Fanuc TP program (LS listing): set_pass_sr.ls

/PROG  SET_PASS_SR
/ATTR
OWNER		= MNEDITOR;
COMMENT		= "";
PROG_SIZE	= 148;
CREATE		= DATE 25-08-01  TIME 09:50:32;
MODIFIED	= DATE 25-08-01  TIME 09:50:32;
FILE_NAME	= ;
VERSION		= 0;
LINE_COUNT	= 1;
MEMORY_SIZE	= 516;
PROTECT		= READ_WRITE;
TCD:  STACK_SIZE	= 0,
      TASK_PRIORITY	= 50,
      TIME_SLICE	= 0,
      BUSY_LAMP_OFF	= 0,
      ABORT_REQUEST	= 0,
      PAUSE_REQUEST	= 0;
DEFAULT_GROUP	= 1,*,*,*,*;
CONTROL_CODE	= 00000000 00000000;
LOCAL_REGISTERS	= 0,0,0;
/MN
   1:  SR[24]=AR[1]    ;
/POS
/END
